{attribute 'analysis' := '-33'}
PROGRAM INTERNAL PRG_RoundTripRepeatedFieldTests
VAR
{IF defined (UNIT_TEST)}
	fbRoundTripRepeatedFieldUInt32Tests		: FB_RoundTripRepeatedFieldUInt32Tests;
	fbRoundTripRepeatedFieldUInt64Tests		: FB_RoundTripRepeatedFieldUInt64Tests;
	fbRoundTripRepeatedFieldStringTests		: FB_RoundTripRepeatedFieldStringTests;
{END_IF}
END_VAR

END_PROGRAM

(* stored: Version 1.1.0.1
   POU PRG_RoundTripRepeatedFieldTests: Id {20818748-fb2b-49f4-acb2-2e9fa6fc3cf8}, SpecialFunc None *)
